INTERFACE I_Brake EXTENDS I_Outputs

PROPERTY AxisState : MC_AxisStates
SET
END_SET
END_PROPERTY

PROPERTY BrakeMode : E_StageBrakeMode
GET
END_GET
SET
END_SET
END_PROPERTY

PROPERTY BrakeRelease : BOOL
GET
END_GET
END_PROPERTY

END_INTERFACE

(* stored: Version 1.1.0.1
   Itf I_Brake: Id {2fdedca0-5e5a-409f-9adf-ce2c06cc3a8d}
   Property AxisState: Id {ba097a17-7813-4cd5-8d3b-6799b9ffbe35}
   Set Set: Id {9a8f1506-33fb-4c48-81ee-5f7bf42268fa}
   Property BrakeMode: Id {bc3ee5d0-39c0-4532-b6ec-0f218e94da1d}
   Get Get: Id {bb8eee33-95ff-47b4-ae9c-75dfd9e983cc}
   Set Set: Id {5ef7ad5b-660a-44fd-9989-042719c95522}
   Property BrakeRelease: Id {d596e907-6a18-4f27-ae07-5b2cff71925d}
   Get Get: Id {cb57d797-17ac-4557-972a-6f4a4092e8eb} *)
